{attribute 'pack_mode' := '1'}
    {attribute 'OPC.UA.DA' := '1'}
    {attribute 'OPC.UA.DA.StructuredType' := '1'}
    (*
    ST_RW_Int_MB_HMI_IgnitionExp
    ==================================================
    Generated from Ignition UDT: RW_Int_MB
    Total tags: 1
    Generated on: 2025-09-15 13:03:45
    *)
    TYPE ST_RW_Int_MB_HMI_IgnitionExp :
    STRUCT
        {attribute 'OPC.UA.DA' := '1'}
        {attribute 'OPC.UA.DA.Description' := '{Description}'}
        // {Description}
        Value : DINT := 0;
    END_STRUCT
    END_TYPE

(* stored: Version 1.1.0.1
   DUT ST_RW_Int_MB_HMI_IgnitionExp: Id {45c5e358-acf5-44ff-9b2c-681f968171af} *)
